DATA_BLOCK "InstDeserializeRows"
{ DB_Accessible_From_OPC_UA := 'FALSE' ;
 S7_Optimized_Access := 'TRUE' }
VERSION : 0.1
NON_RETAIN
"DeserializeRows"

BEGIN

END_DATA_BLOCK

